# EPICS autosave request: energyApp/Db/energy_2BM_settings.req
# This file is used by autosave to determine what PVs to save
# It is also used by txmOptics to determine what PVs to create

# This is the file for the tomoscan_2bm derived class.

#########
# Filters
#########

$(P)$(R)Filters

###############
# Energy change
###############

$(P)$(R)EnergyChoice
